// TIA Portal V16 export
// export: Created 2024-12-03T15:41:45.0755437Z, ExportSetting WithReadOnly, DisplayName Totally Integrated Automation Portal, DisplayVersion V16 Update 6, DisplayName TIA Portal Version Control Interface, DisplayVersion V16 Update 2, DisplayName TIA Portal Openness, DisplayVersion V16 Update 6, DisplayName TIA Portal Teamcenter Gateway, DisplayVersion V16, DisplayName SINAMICS Startdrive Advanced, DisplayVersion V16 Update 5, DisplayName SINAMICS Startdrive G130, G150, S120, S150, SINAMICS MV, S210, DisplayVersion V16 Update 5, DisplayName SINAMICS Startdrive G110M, G120, G120C, G120D, G120P, G115D, DisplayVersion V16 Update 5, DisplayName STEP 7 Professional, DisplayVersion V16 Update 6, DisplayName STEP 7 Safety, DisplayVersion V16, DisplayName WinCC Advanced / Unified PC, DisplayVersion V16 Update 6
TYPE "FLOWSORT_TWISTER_UDT"
// stored: CreationDate 2021-07-13T07:41:36.2278727Z, InterfaceModifiedDate 2020-06-25T06:45:07.2575166Z, IsConsistent true, LibraryConformanceStatus The object is library-conformant., ModifiedDate 2021-03-27T07:36:47.6557293Z
   STRUCT
      Cmd : Struct
         Reset : Bool;
         Interlock : Bool;
         Home_Init { ExternalVisible := 'False'} : Bool;
         SetPointDegAuto : Real;   // The setpoint in degrees
         SetPointDegManual : Real;
         SpeedServo : Int := 1250;   // mm/sec
         SpeedInit : Int := 10;
         BrakeMode : Word := 16#3;   // The Break mode of the MDR . 1 = "Normal" / 2 = "Free" / 3 ="Servo break"
         Accel : Int := 40;   // The Break mode of the MDR . 1 = "Normal" / 2 = "Free" / 3 ="Servo break"
         Deaccel : Int := 100;   // The speed of the MDR in m/s*1000 .The allowed values depend on the Speed code of the MDR .
         ServoResetPulseCount { ExternalVisible := 'False'} : Bool;   // Set pulse count (position) to zero
         ServoRunToSetpoint { ExternalVisible := 'False'} : Bool;   // Run motor from current pulse count to setpoint
         ServoControlDistance : Int;   // The new position to travel to
      END_STRUCT;
      Alarms : Struct   // Alarms
         MdrAlarms { S7_SetPoint := 'True'} : "ConveyLinxAlarms";
         TimedOutHoming : "HmiAlarm";   // The transfer unit did not received the up feedback in time
         Status : Word;
      END_STRUCT;
      Status : Struct
         Interlocked : Bool;
         ManualModeActive : Bool;
         ManualCommandsDisabled : Bool;
         Running : Bool;
         Homed_Intialized : Bool;
         ActualSpeed : Int;
         ServoStatus : Struct
            LastServoCommandExecuted { ExternalVisible := 'False'} : Bool;
            ResetPulseCount_Echo { ExternalVisible := 'False'} : Bool;
            RunCommand_Echo { ExternalVisible := 'False'} : Bool;
         END_STRUCT;
         Position : Int;
         PositionDeg : Real;
         Current : Int;   // The current consumed by the Left MDR in miliamperes
         MinVoltage : Int;
         MaxVoltage : Int;
         Voltage : Int;   // The voltage in mv
         Frequency : Int;   // MDR frequency in Hz as measured by the Hall effect sensors
         TeperatureMDR : Byte;   // The temperature of the MDR in degrees Celsius
         TemperatureModule : Byte;   // The temperature of the module in degrees Celsius
         Status : Word;   // lsb 0 interlocked | lsb 1 running | lbs2 manual mode active
      END_STRUCT;
      CalculatedSettings : Struct
         PulsesPerDeg : Real;
      END_STRUCT;
      Settings : Struct
         OffsetDeg : Real := 5.0;
         Default : Real := 0.0;
         Option_1 : Real := 45.0;
         Option_2 : Real := 90.0;
         Option_3 : Real := 0.0;
      END_STRUCT;
      Heartbeat : Bool;   // Toggles every 2 seconds
      StopStatus : Struct
         StopActiveCommandPLC { ExternalVisible := 'False'} : Bool;   // Stop active due to stop command from the PLC
         StopActiveOtherModule { ExternalVisible := 'False'} : Bool;   // Stop condition is active on a module in the ConveyStop group
         StopActiveLostConn { ExternalVisible := 'False'} : Bool;   // Stop is active due to a loss of communication connection
         StopActiveLostPLC { ExternalVisible := 'False'} : Bool;   // Stop active due to a loss of connection with the PLC
      END_STRUCT;
      Info { S7_SetPoint := 'True'} : "MotorInfo";
      Zone : Int;
   END_STRUCT;
END_TYPE
